{attribute addProperty BoxType "EL6861-0000-0016"}
{attribute addProperty Id "CtrlAT %Q*Ctrl_316DEF3D1621Data_OutAT %Q*ARRAY[0 ..127] OF USINT10241280"}
{attribute addProperty CRC "2622652350"}
{attribute addProperty SizeInBites "1040"}
{attribute addProperty SizeInBytes "130"}
TYPE COM_RxPDO_Map_3D77FD34 :
STRUCT
	{attribute addProperty Name "Ctrl"}
	Ctrl AT %Q* : Ctrl_316DEF3D;
	{attribute addProperty Name "Data_Out"}
	Data_Out AT %Q* : ARRAY[0 ..127] OF USINT;
END_STRUCT
END_TYPE

(* stored: Version 1.2.0.0, ProductVersion 3.1.4024.9
   DUT COM_RxPDO_Map_3D77FD34: Id {5ec4d7e9-53e2-440e-9eca-a6290665012e} *)
